{attribute 'linkalways'} 
{attribute 'no_explicit_call' := 'This FB is a CLASS and must be accessed using methods or properties'}
{attribute 'enable_dynamic_creation'}
FUNCTION_BLOCK _HRESULT EXTENDS AliasDatatypeBase
VAR
	localData : HRESULT;
	activeData : REFERENCE TO HRESULT REF= localData;
	aliasBaseDatatype : _DINT(localData);
END_VAR

PROPERTY PUBLIC Address : PVOID
GET
Address := ADR(activeData);
END_GET
END_PROPERTY

METHOD PUBLIC ClearReference
VAR_INPUT
END_VAR
activeData REF= localData;
SetBaseDatatypeReference();
END_METHOD

METHOD PUBLIC Clone : I_Datatype
VAR
    pClone : POINTER TO _HRESULT;
END_VAR
pClone := __NEW(_HRESULT(InitialValue := Value));
Clone := pClone^;
END_METHOD

METHOD FB_init : BOOL
VAR_INPUT
	bInitRetains : BOOL; // if TRUE, the retain variables are initialized (warm start / cold start)
	bInCopyCode : BOOL;  // if TRUE, the instance afterwards gets moved into the copy code (online change)
	InitialValue : HRESULT;
END_VAR
localData := InitialValue;
SetBaseDatatypeReference();
AddBaseDatatype(aliasBaseDatatype);
END_METHOD

PROPERTY PUBLIC Identifier : T_MAXSTRING
GET
Identifier := 'HRESULT';
END_GET
END_PROPERTY

METHOD PUBLIC MakeReferenceTo
VAR_INPUT
	ReferenceTarget : REFERENCE TO HRESULT;
END_VAR
activeData REF= ReferenceTarget;
SetBaseDatatypeReference();
END_METHOD

METHOD PROTECTED SetBaseDatatypeReference
VAR_INPUT
END_VAR
aliasBaseDatatype.MakeReferenceTo(activeData);
END_METHOD

PROPERTY PUBLIC Size : UDINT
GET
Size := SIZEOF(activeData);
END_GET
END_PROPERTY

METHOD TryMakeReferenceTo : BOOL
VAR_INPUT
	Target : I_Datatype;
END_VAR
VAR
	targetAsAlias : I_AliasDatatype;
	pTargetData : POINTER TO HRESULT;
END_VAR
IF NOT Target.TryResolveAsAliasDatatype(targetAsAlias) THEN
	RETURN;
END_IF

IF targetAsAlias.Identifier <> Identifier THEN
	RETURN;
END_IF

pTargetData := Target.Address;
activeData REF= pTargetData^;
SetBaseDatatypeReference();
TryMakeReferenceTo := TRUE;
END_METHOD

PROPERTY PUBLIC Value : REFERENCE TO HRESULT
GET
Value REF= activeData;
END_GET
END_PROPERTY

END_FUNCTION_BLOCK

(* stored: Version 1.1.0.1, ProductVersion 3.1.4024.12
   POU _HRESULT: Id {2195aa73-ea85-0370-22e7-b8b77b0cb3d8}, SpecialFunc None
   Folder Constructor: Id {8d74f2c6-4182-0f05-042d-0554c4684118}
   Folder Protected: Id {7349e936-984c-02e2-2dc3-c8b0d1e3f7ff}
   Property Address: Id {8c82dcbc-965c-017c-33c8-347d356958fb}
   Get Get: Id {d0a7fd4c-a671-0431-0369-fbbbc82df2ee}
   Method ClearReference: Id {6c19d87c-3793-0f4f-0a83-ab34eea9037a}
   Method Clone: Id {de01f346-3f03-0e4e-10b8-00f849bd3a38}
   Method FB_init: Id {cac580ad-6e63-0b2d-1309-598512198ff7}
   Property Identifier: Id {92fefe99-7dce-0230-149f-e3daaddb0b62}
   Get Get: Id {42d4700a-4d0b-0b5e-0eb2-d10948dab8d4}
   Method MakeReferenceTo: Id {da4f2811-9020-0ece-0298-44832c64da90}
   Method SetBaseDatatypeReference: Id {c40e7a27-92cb-0f48-03ee-a3252b0f422d}
   Property Size: Id {fc48ea4c-1355-0abc-2a87-fc909b7cc270}
   Get Get: Id {30d2773c-825b-0b7d-1401-b01706c4fe8c}
   Method TryMakeReferenceTo: Id {1d040142-872a-0fa8-1431-7a5681b40fcc}
   Property Value: Id {359d8df8-9a2d-0f45-3774-be1eaf094541}
   Get Get: Id {f01bebe5-9e05-01cb-3125-8ec7613b5dcf} *)
